PROGRAM MAIN
VAR
END_VAR

END_PROGRAM

(* stored: Version 1.1.0.1
   POU MAIN: Id {89e3bc44-e1be-490c-8163-0f3fc0309efe} *)
